TYPE DigitalInputBase_50022E7B :
STRUCT
END_STRUCT
END_TYPE

(* stored: Version 1.2.0.0, ProductVersion 3.1.4024.9
   DUT DigitalInputBase_50022E7B: Id {9a5d2807-304e-413c-9810-53eaf5f0d46e} *)
